PROGRAM Ablauf_3530
VAR
    // TODO: lokale Variablen fuer den Ablauf deklarieren
END_VAR


// TODO: Hauptprogramm-Code fuer Ablauf hier einfuegen


METHOD M_VisuKomm : BOOL
VAR_INPUT
    Nr          : INT;
END_VAR
VAR_IN_OUT
    anVisu      : INT;
    vonVisu     : INT;
END_VAR

VAR_INST
    result                  : INT;
    ton_DatenUngueltig      : TON;
    ton_DatenTimeout        : TON;
    sc                      : INT;
END_VAR

// Schnistelle zur VISU Kommunikation
// Starttrigger belegen als Antwort wird auf die 5= gut oder 9=schlecht gewartet.
// Kommunikationstimeout nach 5 Sekunden und wird automatisch wieder neugestartet

ton_DatenTimeout(IN:= anVisu <> 0 AND vonVisu = 0, PT:=T#3S);
ton_DatenUngueltig(IN:= sc = 20, PT:=T#500MS);

CASE sc OF
    0:  // Anfrage starten und auf Antwort warten
        anVisu := Nr;
        result := 0;
        IF vonVisu <> 0 THEN
            IF (vonVisu MOD Nr) = 5 THEN
                sc := 10;
            ELSIF (vonVisu MOD Nr) = 9 THEN
                sc := 20;
            END_IF
        ELSIF ton_DatenTimeout.Q THEN
            sc := 20;
        END_IF

    10: // Antwort 5 erhalten
        anVisu := 0;
        IF vonVisu = 0 THEN
            M_VisuKomm := TRUE;
            result := 1;
            sc := 0;
        END_IF

    20: // Timeout, 1 Sekunde warten und erneut antriggern
        IF ton_DatenUngueltig.Q THEN
            anVisu := 0;
            IF vonVisu = 0 THEN
                result := -1;
                sc := 0;
            END_IF
        END_IF

END_CASE
END_METHOD


METHOD M_VisuKommInt : INT
VAR_INPUT
    Nr          : INT;
END_VAR
VAR_IN_OUT
    anVisu      : INT;
    vonVisu     : INT;
END_VAR

VAR_INST
    result                  : INT;
    ton_DatenUngueltig      : TON;
    ton_DatenTimeout        : TON;
    sc                      : INT;
END_VAR

// Schnistelle zur VISU Kommunikation
// Starttrigger belegen als Antwort wird auf die 5= gut oder 9=schlecht gewartet.
// Kommunikationstimeout nach 5 Sekunden und wird automatisch wieder neugestartet

ton_DatenTimeout(IN:= anVisu <> 0 AND vonVisu = 0, PT:=T#3S);
ton_DatenUngueltig(IN:= anVisu = 0 AND vonVisu = 0, PT:=T#500MS);

CASE sc OF
    0:  // Anfrage starten und auf Antwort warten
        anVisu := Nr;
        result := 0;
        IF vonVisu <> 0 THEN
            IF (vonVisu MOD Nr) = 5 THEN
                sc := 10;
            ELSIF (vonVisu MOD Nr) = 9 THEN
                sc := 15;
            END_IF
        ELSIF ton_DatenTimeout.Q THEN
            sc := 20;
        END_IF

    10: // Antwort 5 erhalten (OK)
        anVisu := 0;
        IF vonVisu = 0 THEN
            M_VisuKommInt := 1;
            result := 1;
            sc := 0;
        END_IF

    15: // Antwort 9 erhalten (Fehler)
        anVisu := 0;
        IF vonVisu = 0 THEN
            M_VisuKommInt := -1;
            result := 1;
            sc := 0;
        END_IF

    20: // Timeout, 1 Sekunde warten und erneut antriggern
        anVisu := 0;
        IF vonVisu = 0 THEN
            result := -1;
            IF ton_DatenUngueltig.Q THEN
                sc := 0;
            END_IF
        END_IF

END_CASE
END_METHOD

END_PROGRAM

(* stored: Version 1.1.0.1
   POU Ablauf_3530: Id {c34c7a80-8362-4489-9555-5a1ef5e61c4e}, SpecialFunc None
   Method M_VisuKomm: Id {1f767fdc-c514-472d-a9ac-f0746cd07596}
   Method M_VisuKommInt: Id {c1b02cbc-5b00-46ac-aae1-079be0ad3ba1} *)
